FUNCTION_BLOCK CT_ReactorActual (* Basic Function Block Type *)
  (* Standard: 61499-2 *)
  (* Version 0.0, 7/5/2026, Schneider Electric, Template *)
  PACKAGE SE.Nereda;
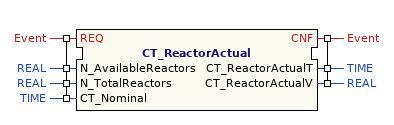
  EVENT_INPUT
    REQ WITH N_AvailableReactors, N_TotalReactors, CT_Nominal; (* Normal Execution Request *)
  END_EVENT
  EVENT_OUTPUT
    CNF WITH CT_ReactorActualT, CT_ReactorActualV; (* Execution Confirmation *)
  END_EVENT
  VAR_INPUT
    N_AvailableReactors : REAL;
    N_TotalReactors : REAL;
    CT_Nominal : TIME;
  END_VAR
  VAR_OUTPUT
    CT_ReactorActualT : TIME;
    CT_ReactorActualV : REAL;
  END_VAR
  VAR
    InCT_Nominal : REAL;
    InCT_ReactorActual : REAL;
  END_VAR
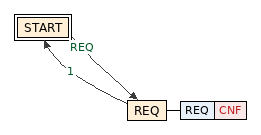
  EC_STATES
    START; (* Initial State *)
    REQ : REQ -> CNF; (* Normal execution *)
  END_STATES
  EC_TRANSITIONS
    START TO REQ := REQ;
    REQ TO START := 1;
  END_TRANSITIONS
  ALGORITHM REQ IN ST: (* Normally executed algorithm *)
;
InCT_Nominal := TIME_TO_REAL(CT_Nominal);

IF N_TotalReactors > 0.0 THEN
	InCT_ReactorActual := (N_AvailableReactors / N_TotalReactors) * InCT_Nominal;
	CT_ReactorActualV := InCT_ReactorActual;
	CT_ReactorActualT := REAL_TO_TIME(InCT_ReactorActual);
ELSE
	CT_ReactorActualV := 0;
	CT_ReactorActualT := T#0s;
END_IF;
  END_ALGORITHM
END_FUNCTION_BLOCK
